# EPICS autosave request: SR570/sr570_settings.req
$(P)M1:Gain:Fine-SP.VAL
$(P)M1:Offset:Fine-SP.VAL
$(P)M1:Bias-SP.VAL
$(P)M1:Mode:Cal-Sel.VAL
$(P)M1:Offset-Sel.VAL
$(P)M1:Offset:Cal-Sel.VAL
$(P)M1:Offset:Sign-Sel.VAL
$(P)M1:Bias-Sel.VAL
$(P)M1:Out:Invert-Sel.VAL
$(P)M1:Out:Blank-Sel.VAL
$(P)M1:Gain:Decade-SP.VAL
$(P)M1:Gain:Val-SP.VAL
$(P)M1:Offset:Decade-SP.VAL
$(P)M1:Offset:Val-SP.VAL
$(P)M1:Filter-Sel.VAL
$(P)M1:Filter:Low-Sel.VAL
$(P)M1:Filter:High-Sel.VAL
$(P)M1:Mode:Gain-Sel.VAL
